// TIA Portal V17 export
// export: Created 2023-12-22T15:08:03.5560164Z, ExportSetting WithDefaults, DisplayName Totally Integrated Automation Portal, DisplayVersion V17, DisplayName TIA Portal Openness, DisplayVersion V17, DisplayName TIA Portal Version Control Interface, DisplayVersion V17, DisplayName STEP 7 Professional, DisplayVersion V17, DisplayName STEP 7 Safety, DisplayVersion V17, DisplayName WinCC Advanced, DisplayVersion V17
DATA_BLOCK "Z_1_1_DB"   // DB700
VERSION : 0.1
// stored: AutoNumber false, DBAccessibleFromOPCUA true, DBAccessibleFromWebserver true, InstanceOfName DRV_V_D2, InstanceOfType FB
"DRV_V_D2"
   // VAR_INPUT
   //    All_Block : Bool;
   // END_VAR
   // VAR_IN_OUT
   //    FB_QF : Bool;
   //    FB_KM_Open : Bool;
   //    FB_KM_Close : Bool;
   //    FB_Open : Bool;
   //    FB_Close : Bool;
   //    S_Alarm : Bool;
   //    CMD_Open : Bool;
   //    CMD_Close : Bool;
   // END_VAR
   // VAR RETAIN
   //    CMD : "CMD";
   //    Mode : Int;
   //    Status : Int;
   //    Use : Struct
   //       QF { S7_SetPoint := 'True'} : Bool := FALSE;
   //       KM_Open { S7_SetPoint := 'True'} : Bool := FALSE;
   //       KM_Close { S7_SetPoint := 'True'} : Bool := FALSE;
   //       Open { S7_SetPoint := 'True'} : Bool := TRUE;
   //       Close { S7_SetPoint := 'True'} : Bool := TRUE;
   //       One_KM { S7_SetPoint := 'True'} : Bool := FALSE;
   //       Electro { S7_SetPoint := 'True'} : Bool := TRUE;
   //       Cross { S7_SetPoint := 'True'} : Bool := FALSE;
   //       CMD_Open { S7_SetPoint := 'True'} : Bool := TRUE;
   //       CMD_Close { S7_SetPoint := 'True'} : Bool := TRUE;
   //       CMD_Reset : Bool;
   //       Local_Keys { S7_SetPoint := 'True'} : Bool := FALSE;
   //       Local_EndPoint : Bool;
   //    END_STRUCT;
   //    FB : Struct
   //       QF : Bool;
   //       KM_Open : Bool;
   //       KM_Close : Bool;
   //       Open : Bool;
   //       Close : Bool;
   //       Reserv : Bool;
   //       Local_Open : Bool;
   //       Local_Close : Bool;
   //    END_STRUCT;
   //    ON : Bool;
   //    OFF : Bool;
   //    REQ_Open : Bool;
   //    REQ_Close : Bool;
   //    Tx { S7_SetPoint := 'True'} : Array[0..4] of "Time_S";
   //    Inv : Struct
   //       CMD { S7_SetPoint := 'True'} : Bool := FALSE;
   //       QF { S7_SetPoint := 'True'} : Bool := FALSE;
   //       KM_Open { S7_SetPoint := 'True'} : Bool := FALSE;
   //       KM_Close { S7_SetPoint := 'True'} : Bool := FALSE;
   //       Serivce { S7_SetPoint := 'True'} : Bool := FALSE;
   //       Open { S7_SetPoint := 'True'} : Bool := FALSE;
   //       Close { S7_SetPoint := 'True'} : Bool := FALSE;
   //       Local_Open { S7_SetPoint := 'True'} : Bool := FALSE;
   //       Local_Close { S7_SetPoint := 'True'} : Bool := FALSE;
   //    END_STRUCT;
   //    Alarm : Struct
   //       Block : Bool;
   //       QF : Bool;
   //       KM_Open : Bool;
   //       KM_Close : Bool;
   //       Two_S : Bool;
   //       Open : Bool;
   //       Close : Bool;
   //       OpTime : Bool;
   //       Alarm : Bool;
   //    END_STRUCT;
   //    Alarms : Word;
   //    Events : Word;
   //    pos : Array[0..15] of Bool;
   //    OpTime_h : DInt;
   //    OpTime_s { S7_SetPoint := 'True'} : DInt := 3544;
   //    CodeID { S7_SetPoint := 'True'} : Int := 0;
   //    Indirect : Struct
   //       FB_QF { S7_SetPoint := 'True'} : Bool := TRUE;
   //       FB_KM_Open { S7_SetPoint := 'True'} : Bool := TRUE;
   //       FB_KM_Close { S7_SetPoint := 'True'} : Bool := TRUE;
   //       FB_Open { S7_SetPoint := 'True'} : Bool := TRUE;
   //       FB_Close { S7_SetPoint := 'True'} : Bool := TRUE;
   //       FB_Alarm { S7_SetPoint := 'True'} : Bool := TRUE;
   //       CMD_Open { S7_SetPoint := 'True'} : Bool := TRUE;
   //       CMD_Close { S7_SetPoint := 'True'} : Bool := TRUE;
   //    END_STRUCT;
   //    Indirect_BYTE : Struct
   //       FB_QF { S7_SetPoint := 'True'} : Int := 1;
   //       FB_KM_Open { S7_SetPoint := 'True'} : Int := 0;
   //       FB_KM_Close { S7_SetPoint := 'True'} : Int := 0;
   //       FB_Open { S7_SetPoint := 'True'} : Int := 1;
   //       FB_Close { S7_SetPoint := 'True'} : Int := 2;
   //       FB_Alarm { S7_SetPoint := 'True'} : Int := 2;
   //       CMD_Open { S7_SetPoint := 'True'} : Int := 0;
   //       CMD_Close { S7_SetPoint := 'True'} : Int := 1;
   //       CMD_Reset : Int;
   //    END_STRUCT;
   //    Indirect_BIT : Struct
   //       FB_QF { S7_SetPoint := 'True'} : Int := 6;
   //       FB_KM_Open { S7_SetPoint := 'True'} : Int := 9;
   //       FB_KM_Close { S7_SetPoint := 'True'} : Int := 9;
   //       FB_Open { S7_SetPoint := 'True'} : Int := 7;
   //       FB_Close { S7_SetPoint := 'True'} : Int := 0;
   //       FB_Alarm { S7_SetPoint := 'True'} : Int := 1;
   //       CMD_Open { S7_SetPoint := 'True'} : Int := 7;
   //       CMD_Close { S7_SetPoint := 'True'} : Int := 0;
   //       CMD_Reset : Int;
   //    END_STRUCT;
   // END_VAR
BEGIN
   Tx[0..1].SP := 0;
   Tx[2..3].SP := 150;
   Tx[4].SP := 2;
END_DATA_BLOCK
